{attribute 'GeneratedUsingTerminal: EL1502-0000-0018'}
{attribute addProperty BoxType "EL1502-0000-0018"}
{attribute addProperty Id "CNT_InputsAT %I*CNT_Inputs_B6C38E7112CNT_OutputsAT %Q*CNT_Outputs_458039AE8WcStateAT %I*WcState_9091E0EB2InfoDataAT %I*InfoData_94A18F5E2"}
{attribute addProperty CRC "3158905868"}
{attribute addProperty Size "24"}
TYPE EL1502_BC49140C EXTENDS EtcSlaveTerminalBase_947E5A46 :
STRUCT
	{attribute addProperty Name "CNT_Inputs"}
	CNT_Inputs : CNT_Inputs_B6C38E71;
	{attribute addProperty Name "CNT_Outputs"}
	CNT_Outputs : CNT_Outputs_458039AE;
	{attribute addProperty Name "WcState"}
	WcState : WcState_9091E0EB;
	{attribute addProperty Name "InfoData"}
	InfoData : InfoData_94A18F5E;
END_STRUCT
END_TYPE

(* stored: Version 1.2.0.0, ProductVersion 3.1.4024.9
   DUT EL1502_BC49140C: Id {a1994b7f-300e-4305-9a91-a0bcfcc37f2a} *)
